(* Logix 5000 project; controller Drives_Line1 1756-L72 rev 20.13; software revision 20.04; part 9 of 21 *)
(* tags used below, declared in another part *)
   IO_State_Pinch_2 : INT;
   IO_State_Tmp_Pinch_2 : INT;
   Pinchroll_2_EncRes : DINT;
   Pinchroll_2_FB_Count_Old : DINT;
   Pinchroll_2_Max_FB_Counts : DINT;
   Pinchroll_2_Rev_mm : REAL;
   Pinchroll_2_RPMPerMPS : REAL;
   TonRefOn : TIMER;
   zPinchroll_2_Max_rev : REAL;
   Bridle_01 : UDT_Bridle_3M;
   EntryCtrl : UDT_Control_Zone;
   In_Config : UDT_Config;
   LineCmd : UDT_Commands_Line;
   Out_Feedbacks : UDT_Fdbks;
   Out_Status : UDT_Status;
   Pinchroll_2 : UDT_Pinchroll;
   Pinchroll_2_FB_Difference : DINT;
   Pinchroll_2_FB_Update_Valid : BOOL;
   Pinchroll_2_FBCounts_mm : REAL;
   TaskInterval_ms : DINT;
   TestConfig_Pinchroll_2 : UDT_Config_Pinch;
   Unwinder_1 : UDT_Unwinder;
   Unwinder_2 : UDT_Unwinder;
   zConfigFromMaster : BOOL;
   zPi : REAL;
   zPinchroll_2_EncRes : DINT;
(* P13_Pinchroll_2, continued *)

ROUTINE R03_Drive_Interface   (* ladder *)
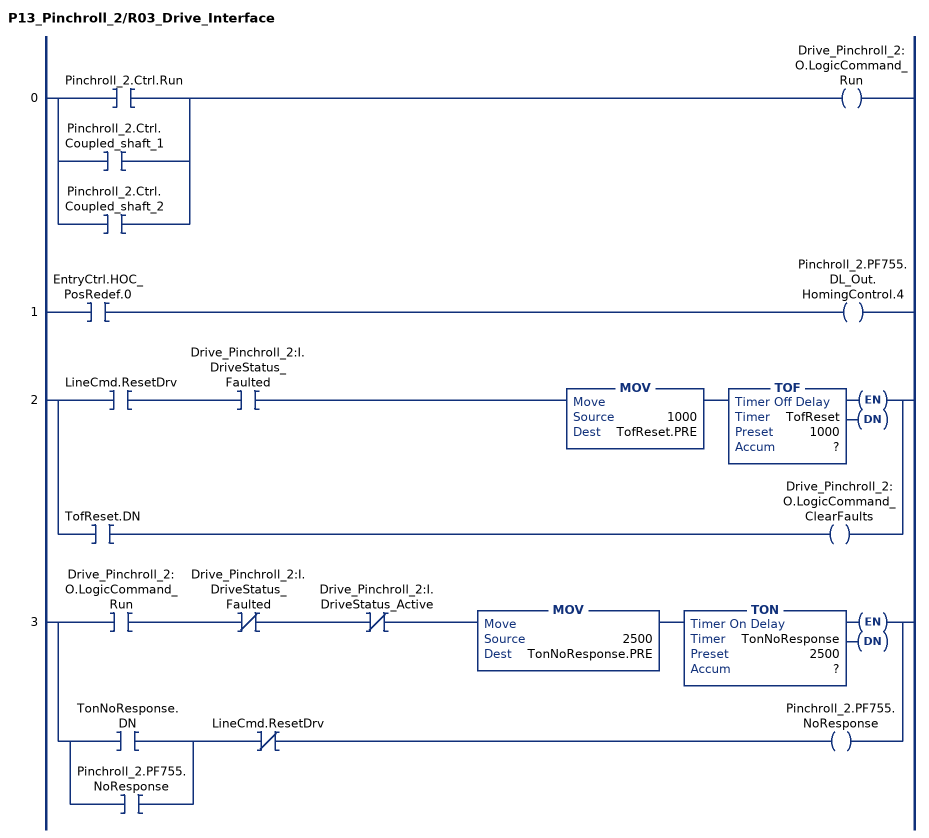
   0: [XIC(Pinchroll_2.Ctrl.Run) ,XIC(Pinchroll_2.Ctrl.Coupled_shaft_1) ,XIC(Pinchroll_2.Ctrl.Coupled_shaft_2) ]OTE(Drive_Pinchroll_2:O.LogicCommand_Run);
   1: XIC(EntryCtrl.HOC_PosRedef.0)OTE(Pinchroll_2.PF755.DL_Out.HomingControl.4);
   2: [XIC(LineCmd.ResetDrv) XIC(Drive_Pinchroll_2:I.DriveStatus_Faulted) MOV(1000,TofReset.PRE) TOF(TofReset,?,?) ,XIC(TofReset.DN) OTE(Drive_Pinchroll_2:O.LogicCommand_ClearFaults) ];
   3: [XIC(Drive_Pinchroll_2:O.LogicCommand_Run) XIO(Drive_Pinchroll_2:I.DriveStatus_Faulted) XIO(Drive_Pinchroll_2:I.DriveStatus_Active) MOV(2500,TonNoResponse.PRE) TON(TonNoResponse,?,?) ,[XIC(TonNoResponse.DN) ,XIC(Pinchroll_2.PF755.NoResponse) ] XIO(LineCmd.ResetDrv) OTE(Pinchroll_2.PF755.NoResponse) ];
END_ROUTINE

ROUTINE R04_State   (* ladder *)
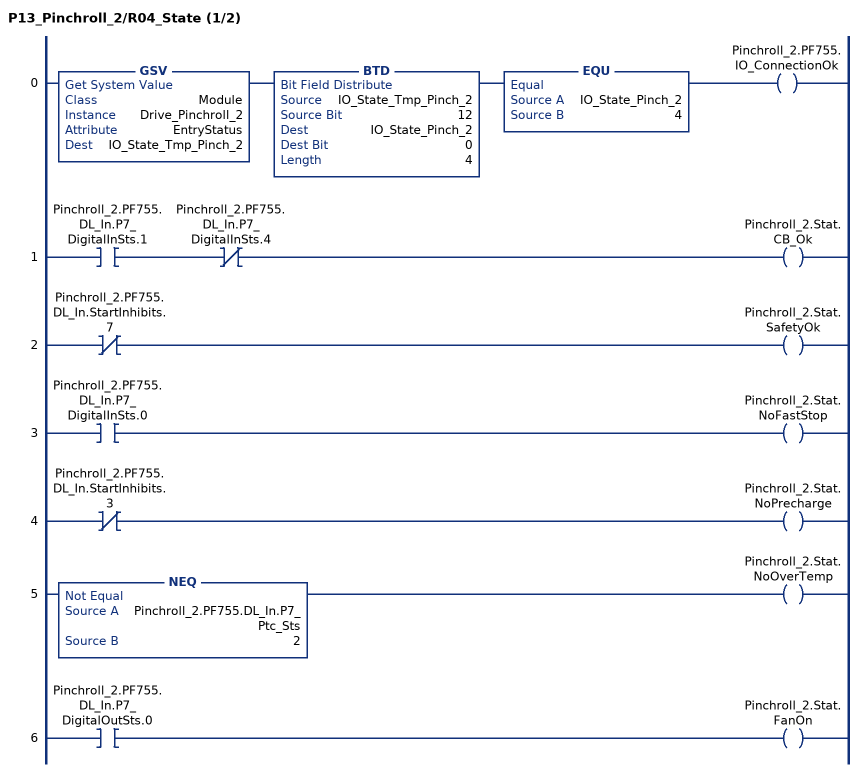
   0: GSV(Module,Drive_Pinchroll_2,EntryStatus,IO_State_Tmp_Pinch_2)BTD(IO_State_Tmp_Pinch_2,12,IO_State_Pinch_2,0,4)EQU(IO_State_Pinch_2,4)OTE(Pinchroll_2.PF755.IO_ConnectionOk);
   1: XIC(Pinchroll_2.PF755.DL_In.P7_DigitalInSts.1)XIO(Pinchroll_2.PF755.DL_In.P7_DigitalInSts.4)OTE(Pinchroll_2.Stat.CB_Ok);
   2: XIO(Pinchroll_2.PF755.DL_In.StartInhibits.7)OTE(Pinchroll_2.Stat.SafetyOk);
   3: XIC(Pinchroll_2.PF755.DL_In.P7_DigitalInSts.0)OTE(Pinchroll_2.Stat.NoFastStop);
   4: XIO(Pinchroll_2.PF755.DL_In.StartInhibits.3)OTE(Pinchroll_2.Stat.NoPrecharge);
   5: NEQ(Pinchroll_2.PF755.DL_In.P7_Ptc_Sts,2)OTE(Pinchroll_2.Stat.NoOverTemp);
   6: XIC(Pinchroll_2.PF755.DL_In.P7_DigitalOutSts.0)OTE(Pinchroll_2.Stat.FanOn);
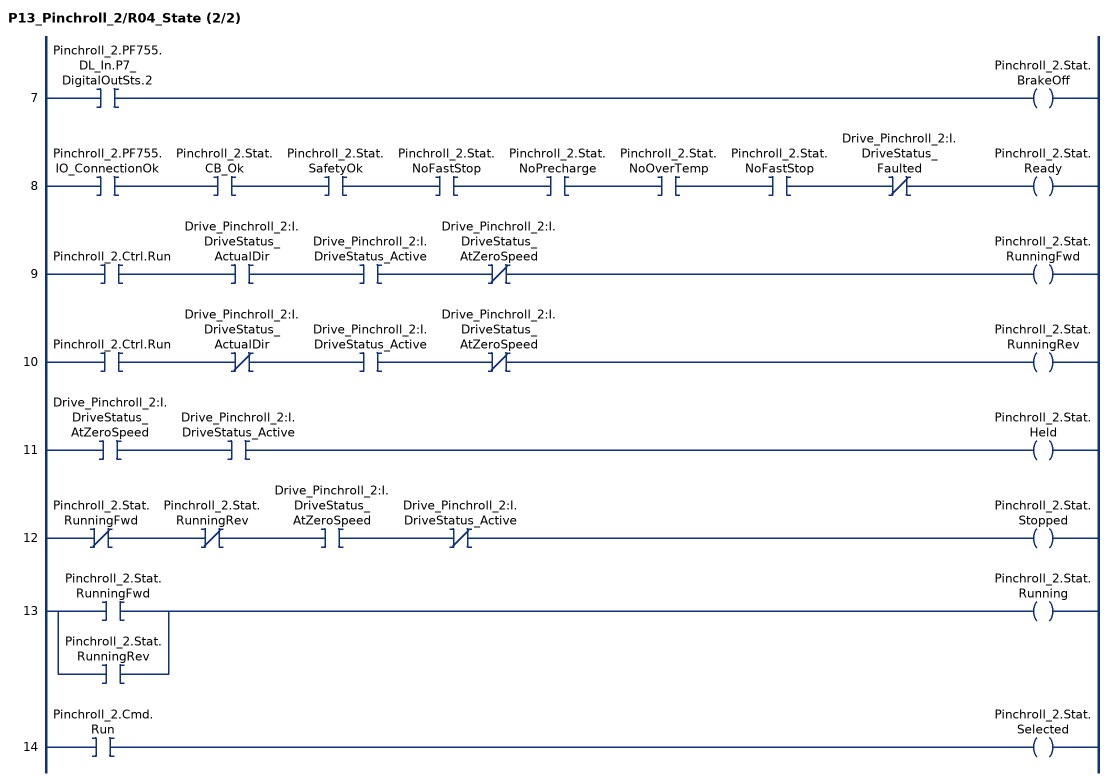
   7: XIC(Pinchroll_2.PF755.DL_In.P7_DigitalOutSts.2)OTE(Pinchroll_2.Stat.BrakeOff);
   8: XIC(Pinchroll_2.PF755.IO_ConnectionOk)XIC(Pinchroll_2.Stat.CB_Ok)XIC(Pinchroll_2.Stat.SafetyOk)XIC(Pinchroll_2.Stat.NoFastStop)XIC(Pinchroll_2.Stat.NoPrecharge)XIC(Pinchroll_2.Stat.NoOverTemp)XIC(Pinchroll_2.Stat.NoFastStop)XIO(Drive_Pinchroll_2:I.DriveStatus_Faulted)OTE(Pinchroll_2.Stat.Ready);
   9: XIC(Pinchroll_2.Ctrl.Run)XIC(Drive_Pinchroll_2:I.DriveStatus_ActualDir)XIC(Drive_Pinchroll_2:I.DriveStatus_Active)XIO(Drive_Pinchroll_2:I.DriveStatus_AtZeroSpeed)OTE(Pinchroll_2.Stat.RunningFwd);
   10: XIC(Pinchroll_2.Ctrl.Run)XIO(Drive_Pinchroll_2:I.DriveStatus_ActualDir)XIC(Drive_Pinchroll_2:I.DriveStatus_Active)XIO(Drive_Pinchroll_2:I.DriveStatus_AtZeroSpeed)OTE(Pinchroll_2.Stat.RunningRev);
   11: XIC(Drive_Pinchroll_2:I.DriveStatus_AtZeroSpeed)XIC(Drive_Pinchroll_2:I.DriveStatus_Active)OTE(Pinchroll_2.Stat.Held);
   12: XIO(Pinchroll_2.Stat.RunningFwd)XIO(Pinchroll_2.Stat.RunningRev)XIC(Drive_Pinchroll_2:I.DriveStatus_AtZeroSpeed)XIO(Drive_Pinchroll_2:I.DriveStatus_Active)OTE(Pinchroll_2.Stat.Stopped);
   13: [XIC(Pinchroll_2.Stat.RunningFwd) ,XIC(Pinchroll_2.Stat.RunningRev) ]OTE(Pinchroll_2.Stat.Running);
   14: XIC(Pinchroll_2.Cmd.Run)OTE(Pinchroll_2.Stat.Selected);
END_ROUTINE

ROUTINE R05_Control   (* ladder *)
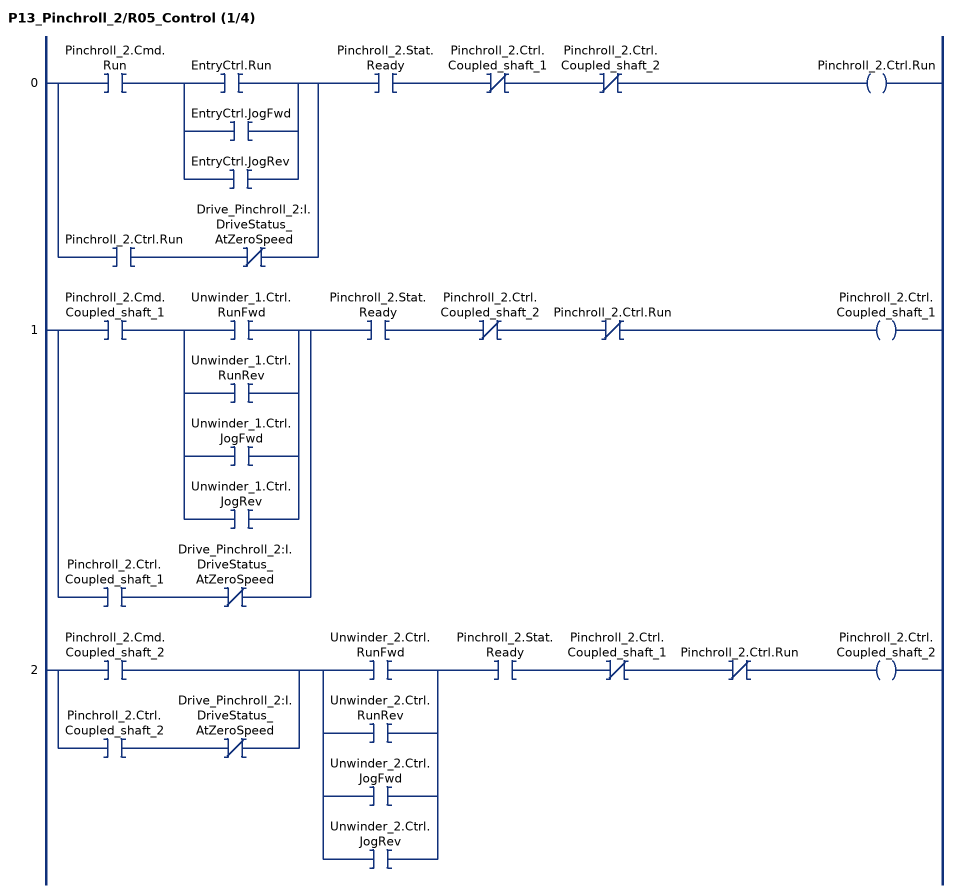
   0: [XIC(Pinchroll_2.Cmd.Run) [XIC(EntryCtrl.Run) ,XIC(EntryCtrl.JogFwd) ,XIC(EntryCtrl.JogRev) ] ,XIC(Pinchroll_2.Ctrl.Run) XIO(Drive_Pinchroll_2:I.DriveStatus_AtZeroSpeed) ]XIC(Pinchroll_2.Stat.Ready)XIO(Pinchroll_2.Ctrl.Coupled_shaft_1)XIO(Pinchroll_2.Ctrl.Coupled_shaft_2)OTE(Pinchroll_2.Ctrl.Run);
   1: [XIC(Pinchroll_2.Cmd.Coupled_shaft_1) [XIC(Unwinder_1.Ctrl.RunFwd) ,XIC(Unwinder_1.Ctrl.RunRev) ,XIC(Unwinder_1.Ctrl.JogFwd) ,XIC(Unwinder_1.Ctrl.JogRev) ] ,XIC(Pinchroll_2.Ctrl.Coupled_shaft_1) XIO(Drive_Pinchroll_2:I.DriveStatus_AtZeroSpeed) ]XIC(Pinchroll_2.Stat.Ready)XIO(Pinchroll_2.Ctrl.Coupled_shaft_2)XIO(Pinchroll_2.Ctrl.Run)OTE(Pinchroll_2.Ctrl.Coupled_shaft_1);
   2: [XIC(Pinchroll_2.Cmd.Coupled_shaft_2) ,XIC(Pinchroll_2.Ctrl.Coupled_shaft_2) XIO(Drive_Pinchroll_2:I.DriveStatus_AtZeroSpeed) ][XIC(Unwinder_2.Ctrl.RunFwd) ,XIC(Unwinder_2.Ctrl.RunRev) ,XIC(Unwinder_2.Ctrl.JogFwd) ,XIC(Unwinder_2.Ctrl.JogRev) ]XIC(Pinchroll_2.Stat.Ready)XIO(Pinchroll_2.Ctrl.Coupled_shaft_1)XIO(Pinchroll_2.Ctrl.Run)OTE(Pinchroll_2.Ctrl.Coupled_shaft_2);
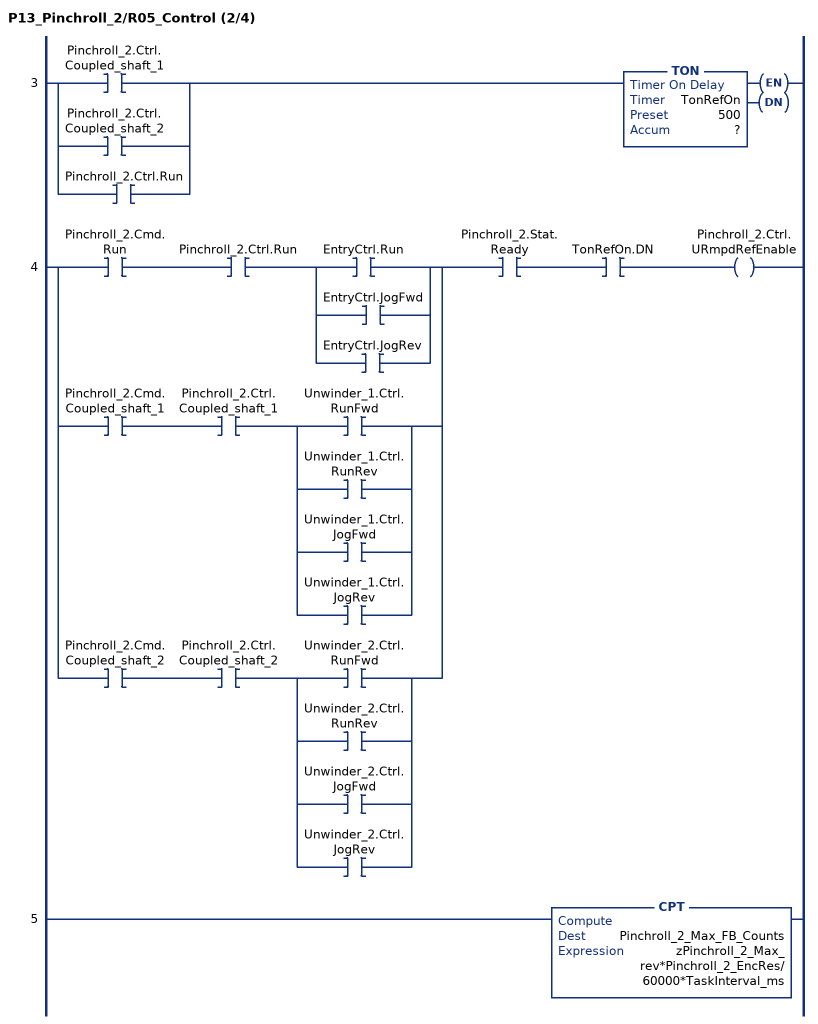
   3: [XIC(Pinchroll_2.Ctrl.Coupled_shaft_1) ,XIC(Pinchroll_2.Ctrl.Coupled_shaft_2) ,XIC(Pinchroll_2.Ctrl.Run) ]TON(TonRefOn,?,?);
   4: [XIC(Pinchroll_2.Cmd.Run) XIC(Pinchroll_2.Ctrl.Run) [XIC(EntryCtrl.Run) ,XIC(EntryCtrl.JogFwd) ,XIC(EntryCtrl.JogRev) ] ,XIC(Pinchroll_2.Cmd.Coupled_shaft_1) XIC(Pinchroll_2.Ctrl.Coupled_shaft_1) [XIC(Unwinder_1.Ctrl.RunFwd) ,XIC(Unwinder_1.Ctrl.RunRev) ,XIC(Unwinder_1.Ctrl.JogFwd) ,XIC(Unwinder_1.Ctrl.JogRev) ] ,XIC(Pinchroll_2.Cmd.Coupled_shaft_2) XIC(Pinchroll_2.Ctrl.Coupled_shaft_2) [XIC(Unwinder_2.Ctrl.RunFwd) ,XIC(Unwinder_2.Ctrl.RunRev) ,XIC(Unwinder_2.Ctrl.JogFwd) ,XIC(Unwinder_2.Ctrl.JogRev) ] ]XIC(Pinchroll_2.Stat.Ready)XIC(TonRefOn.DN)OTE(Pinchroll_2.Ctrl.URmpdRefEnable);
   5: CPT(Pinchroll_2_Max_FB_Counts,zPinchroll_2_Max_rev*Pinchroll_2_EncRes/60000*TaskInterval_ms);
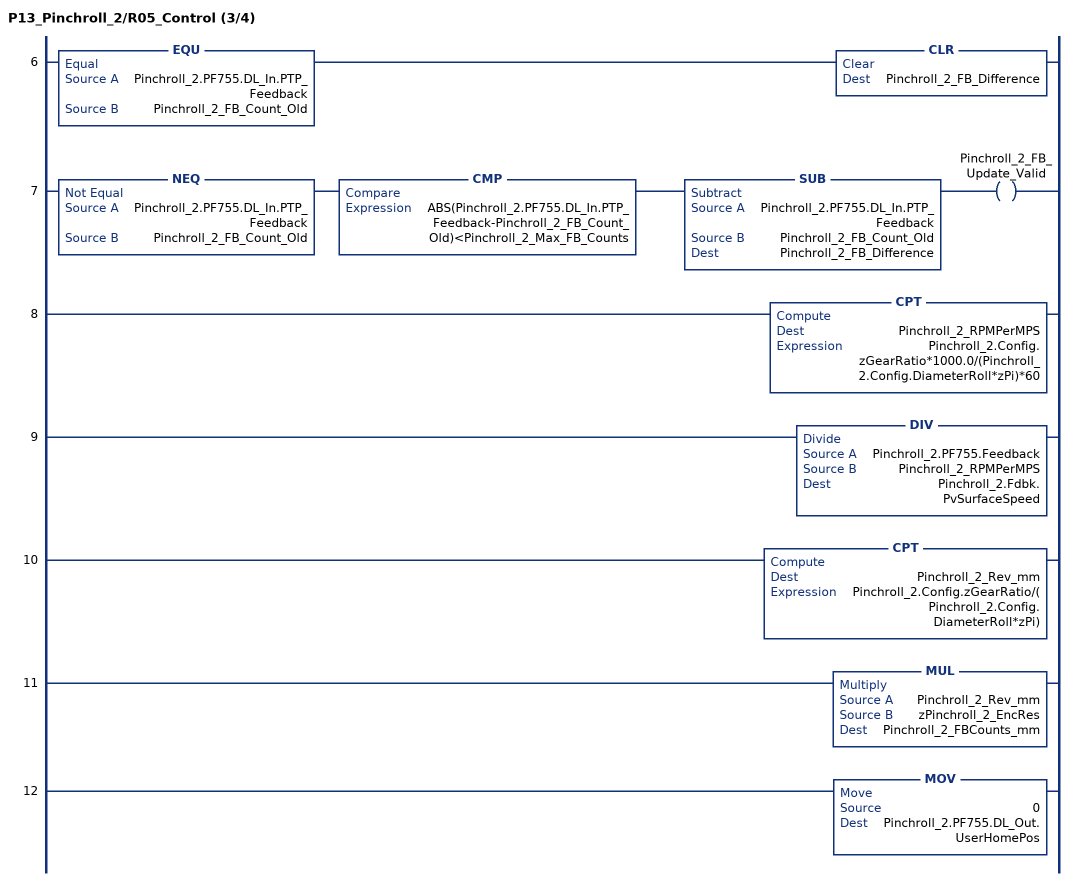
   6: EQU(Pinchroll_2.PF755.DL_In.PTP_Feedback,Pinchroll_2_FB_Count_Old)CLR(Pinchroll_2_FB_Difference);
   7: NEQ(Pinchroll_2.PF755.DL_In.PTP_Feedback,Pinchroll_2_FB_Count_Old)CMP(ABS(Pinchroll_2.PF755.DL_In.PTP_Feedback-Pinchroll_2_FB_Count_Old)<Pinchroll_2_Max_FB_Counts)SUB(Pinchroll_2.PF755.DL_In.PTP_Feedback,Pinchroll_2_FB_Count_Old,Pinchroll_2_FB_Difference)OTE(Pinchroll_2_FB_Update_Valid);
   8: CPT(Pinchroll_2_RPMPerMPS,Pinchroll_2.Config.zGearRatio*1000.0/(Pinchroll_2.Config.DiameterRoll*zPi)*60);
   9: DIV(Pinchroll_2.PF755.Feedback,Pinchroll_2_RPMPerMPS,Pinchroll_2.Fdbk.PvSurfaceSpeed);
   10: CPT(Pinchroll_2_Rev_mm,Pinchroll_2.Config.zGearRatio/(Pinchroll_2.Config.DiameterRoll*zPi));
   11: MUL(Pinchroll_2_Rev_mm,zPinchroll_2_EncRes,Pinchroll_2_FBCounts_mm);
   12: MOV(0,Pinchroll_2.PF755.DL_Out.UserHomePos);
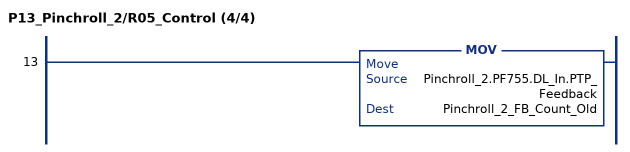
   13: MOV(Pinchroll_2.PF755.DL_In.PTP_Feedback,Pinchroll_2_FB_Count_Old);
END_ROUTINE

ROUTINE R12_DriveRef   (* function block diagram *)
   SHEET 1   // Select speed reference
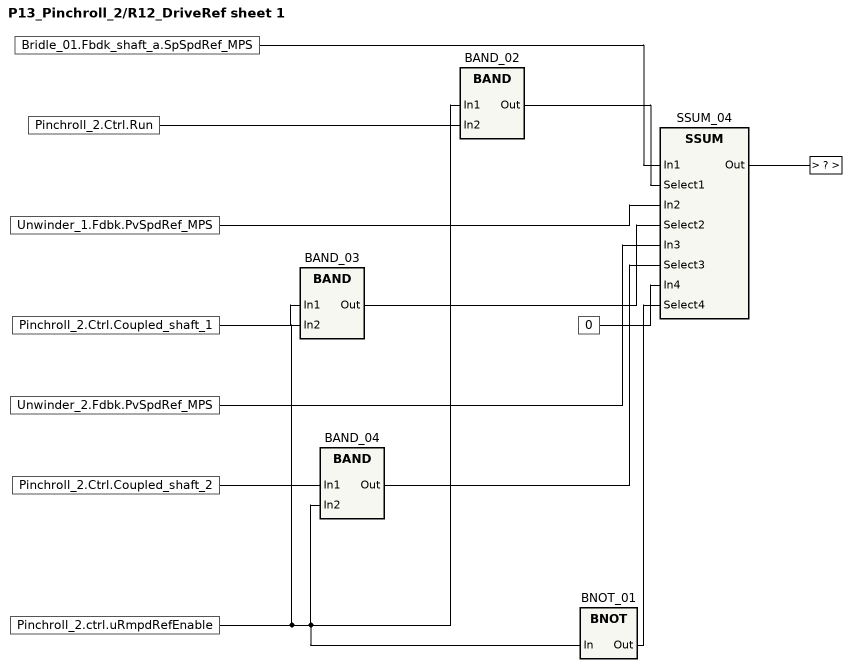
   BAND_03 : BAND(In1 := Pinchroll_2.Ctrl.Coupled_shaft_1, In2 := Pinchroll_2.ctrl.uRmpdRefEnable);
   BAND_04 : BAND(In1 := Pinchroll_2.Ctrl.Coupled_shaft_2, In2 := Pinchroll_2.ctrl.uRmpdRefEnable);
   BAND_02 : BAND(In1 := Pinchroll_2.ctrl.uRmpdRefEnable, In2 := Pinchroll_2.Ctrl.Run);
   BNOT_01 : BNOT(In := Pinchroll_2.ctrl.uRmpdRefEnable);
   SSUM_04 : SSUM(In1 := Bridle_01.Fbdk_shaft_a.SpSpdRef_MPS, Select1 := BAND_02.Out, In2 := Unwinder_1.Fdbk.PvSpdRef_MPS, Select2 := BAND_03.Out, In3 := Unwinder_2.Fdbk.PvSpdRef_MPS, Select3 := BAND_04.Out, In4 := 0, Select4 := BNOT_01.Out);
   WIRE(?) := SSUM_04.Out;
   SHEET 2   // Final speed reference
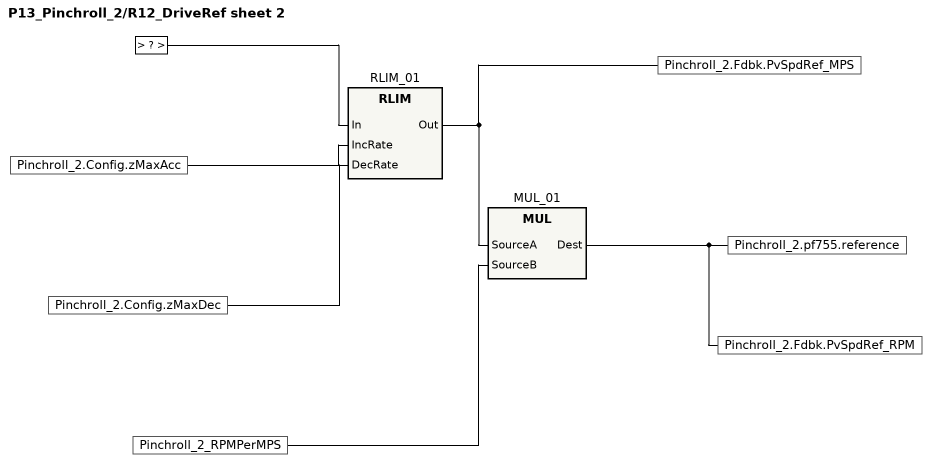
   RLIM_01 : RLIM(In := WIRE(?), IncRate := Pinchroll_2.Config.zMaxAcc, DecRate := Pinchroll_2.Config.zMaxDec);
   MUL_01 : MUL(SourceA := RLIM_01.Out, SourceB := Pinchroll_2_RPMPerMPS);
   Pinchroll_2.Fdbk.PvSpdRef_MPS := RLIM_01.Out;
   Pinchroll_2.Fdbk.PvSpdRef_RPM := MUL_01.Dest;
   Pinchroll_2.pf755.reference := MUL_01.Dest;
   SHEET 3   // Speed reference synchronized
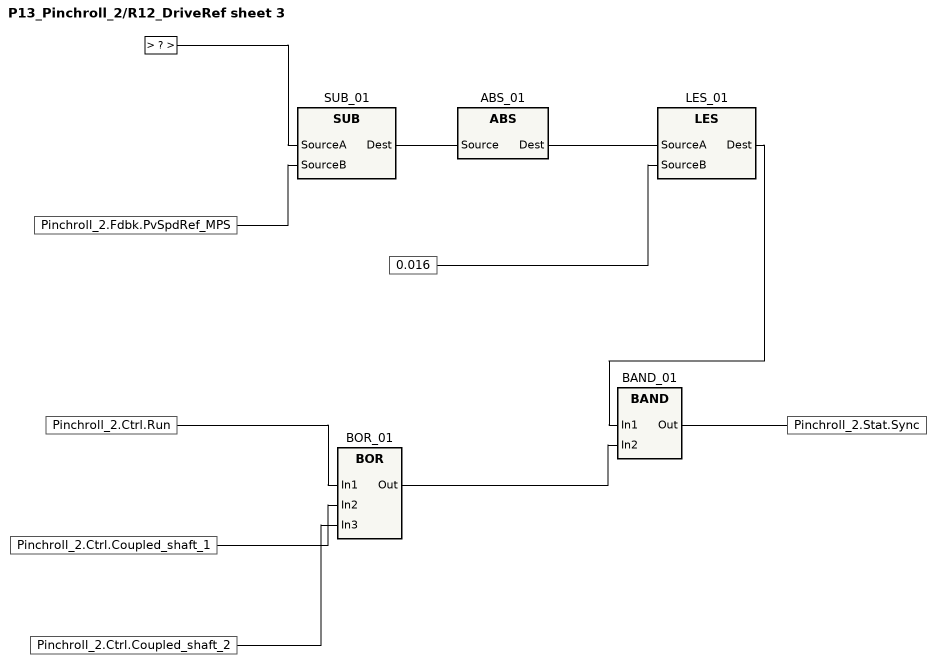
   SUB_01 : SUB(SourceA := WIRE(?), SourceB := Pinchroll_2.Fdbk.PvSpdRef_MPS);
   BOR_01 : BOR(In1 := Pinchroll_2.Ctrl.Run, In2 := Pinchroll_2.Ctrl.Coupled_shaft_1, In3 := Pinchroll_2.Ctrl.Coupled_shaft_2);
   ABS_01 : ABS(Source := SUB_01.Dest);
   LES_01 : LES(SourceA := ABS_01.Dest, SourceB := 0.016);
   BAND_01 : BAND(In1 := LES_01.Dest, In2 := BOR_01.Out);
   Pinchroll_2.Stat.Sync := BAND_01.Out;
END_ROUTINE

ROUTINE R98_ToDrive   (* ladder *)
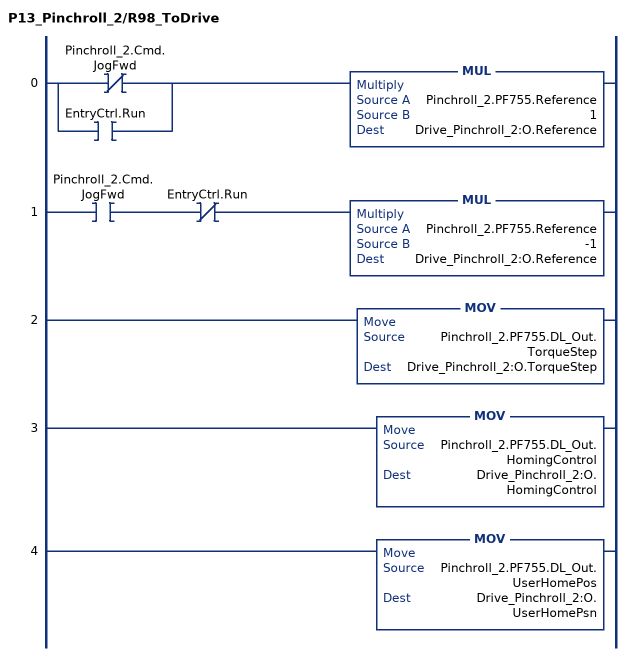
   0: [XIO(Pinchroll_2.Cmd.JogFwd) ,XIC(EntryCtrl.Run) ]MUL(Pinchroll_2.PF755.Reference,1,Drive_Pinchroll_2:O.Reference);
   1: XIC(Pinchroll_2.Cmd.JogFwd)XIO(EntryCtrl.Run)MUL(Pinchroll_2.PF755.Reference,-1,Drive_Pinchroll_2:O.Reference);
   2: MOV(Pinchroll_2.PF755.DL_Out.TorqueStep,Drive_Pinchroll_2:O.TorqueStep);
   3: MOV(Pinchroll_2.PF755.DL_Out.HomingControl,Drive_Pinchroll_2:O.HomingControl);
   4: MOV(Pinchroll_2.PF755.DL_Out.UserHomePos,Drive_Pinchroll_2:O.UserHomePsn);
END_ROUTINE

ROUTINE R999_Test   (* ladder *)
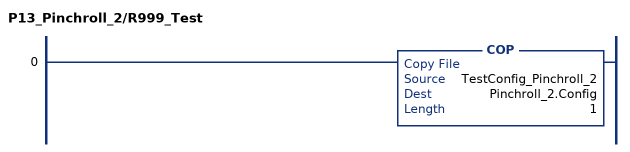
   0: COP(TestConfig_Pinchroll_2,Pinchroll_2.Config,1);
END_ROUTINE

ROUTINE R99_To_Master   (* ladder *)
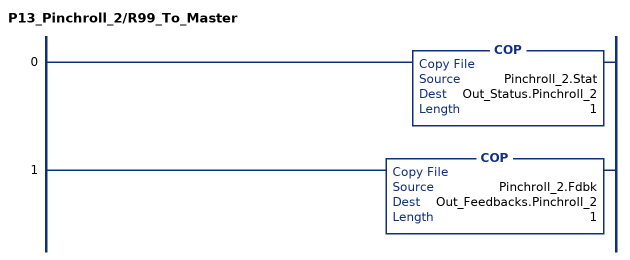
   0: COP(Pinchroll_2.Stat,Out_Status.Pinchroll_2,1);
   1: COP(Pinchroll_2.Fdbk,Out_Feedbacks.Pinchroll_2,1);
END_ROUTINE
END_PROGRAM

PROGRAM P14_Bridle_01   (* main routine R00_Main *)
VAR
   ADD_01 : FBD_MATH;
   BNOT_01 : FBD_BOOLEAN_NOT := (Out := 1);
   BNOT_02 : FBD_BOOLEAN_NOT := (In := 1);
   BNOT_03 : FBD_BOOLEAN_NOT := (Out := 1);
   Bridle_01_FB_Count_Old : DINT := 9220666;
   Bridle_01_Max_FBcounts : REAL := 5120.0;
   Bridle_01_SpdTrimMPS : REAL;
   Bridle_01_SpdTrimPct : REAL;
   Bridle_01a_RPMPerMPS : REAL := 3085.579;
   Bridle_01b_RPMPerMPS : REAL := 3085.579;
   Bridle_01c_RPMPerMPS : REAL := 2634.4192;
   DIV_01 : FBD_MATH := (SourceB := 100.0);
   EQU_01 : FBD_COMPARE := (SourceA := 0.08467744);
   IO_State_Bridle_01a : INT := 4;
   IO_State_Bridle_01b : INT := 4;
   IO_State_Bridle_01c : INT := 4;
   IO_State_Tmp_Bridle_01a : INT := 16384;
   IO_State_Tmp_Bridle_01b : INT := 16384;
   IO_State_Tmp_Bridle_01c : INT := 16384;
   MUL_01 : FBD_MATH := (SourceB := 3085.579);
   MUL_02 : FBD_MATH := (SourceB := 3085.579);
   MUL_05 : FBD_MATH;
   MUL_06 : FBD_MATH := (SourceB := 2634.4192);
   Ons : DINT;
   PI_02 : PROP_INT := (In := -2.3841858e-07, Initialize := 1, Kp := 0.1, Wld := 0.01, HighLimit := 2.5, LowLimit := -2.5, ShapeKpPlus := 1.0, ShapeKpMinus := 1.0, ShapeWldPlus := 1.0, ShapeWldMinus := 1.0, RTSTime := 1, DeltaT := 0.05);
   PulsReset_PID : TIMER := (PRE := 250);
   SCL_09 : SCALE := (InRawMax := 100.0, InRawMin := -100.0, InEUMax := 2.5, InEUMin := -2.5, Limiting := 1, Out := -2.3841858e-07);
   SUB_02 : FBD_MATH;
   TimeOn_PIDOn : TIMER := (PRE := 500);
   TofReset : TIMER := (PRE := 1000, ACC := 1000);
   TonNoResponse : TIMER[3] := ([0].PRE := 2500, [1].PRE := 2500, [2].PRE := 2500);
   zBridle_01_Ki_SpdTrim : REAL := 0.01;
   zBridle_01_Kp_SpdTrim : REAL := 0.1;
   zBridle_01_Max_rev : DINT := 1500;
   zBridle_01_MaxTrimSpdTrim : REAL := 2.5;
   zBridle_01_MinTrimSpdTrim : REAL := -2.5;
   zBridle_01b_EncRes : REAL := 4096.0;
END_VAR

ROUTINE R00_Main   (* ladder *)
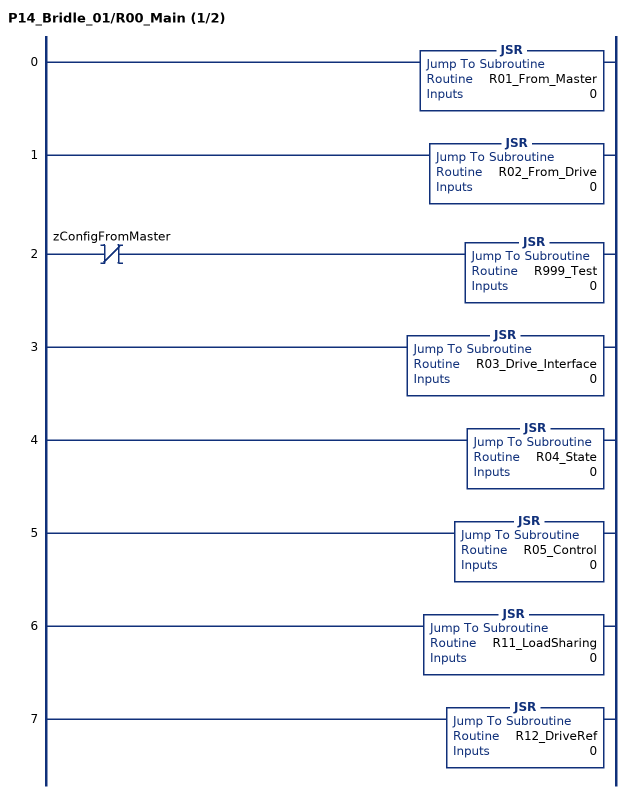
   0: JSR(R01_From_Master,0);
   1: JSR(R02_From_Drive,0);
   2: XIO(zConfigFromMaster)JSR(R999_Test,0);
   3: JSR(R03_Drive_Interface,0);
   4: JSR(R04_State,0);
   5: JSR(R05_Control,0);
   6: JSR(R11_LoadSharing,0);
   7: JSR(R12_DriveRef,0);
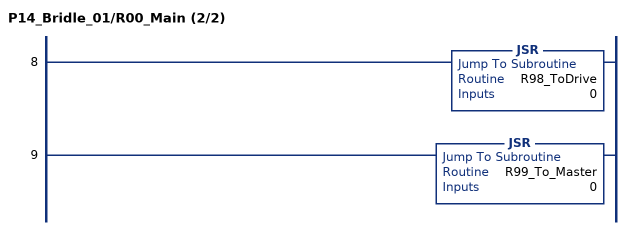
   8: JSR(R98_ToDrive,0);
   9: JSR(R99_To_Master,0);
END_ROUTINE

ROUTINE R01_From_Master   (* ladder *)
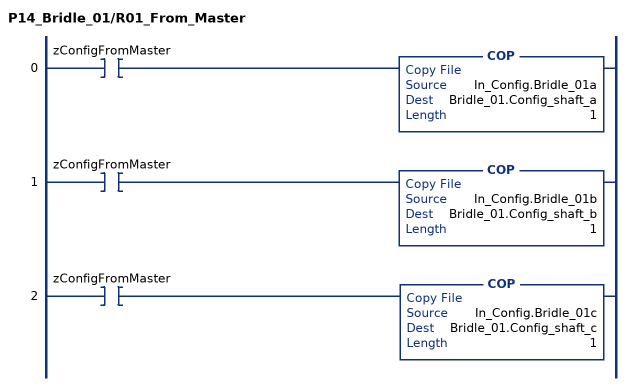
   0: XIC(zConfigFromMaster)COP(In_Config.Bridle_01a,Bridle_01.Config_shaft_a,1);
   1: XIC(zConfigFromMaster)COP(In_Config.Bridle_01b,Bridle_01.Config_shaft_b,1);
   2: XIC(zConfigFromMaster)COP(In_Config.Bridle_01c,Bridle_01.Config_shaft_c,1);
END_ROUTINE

ROUTINE R02_From_Drive   (* ladder *)
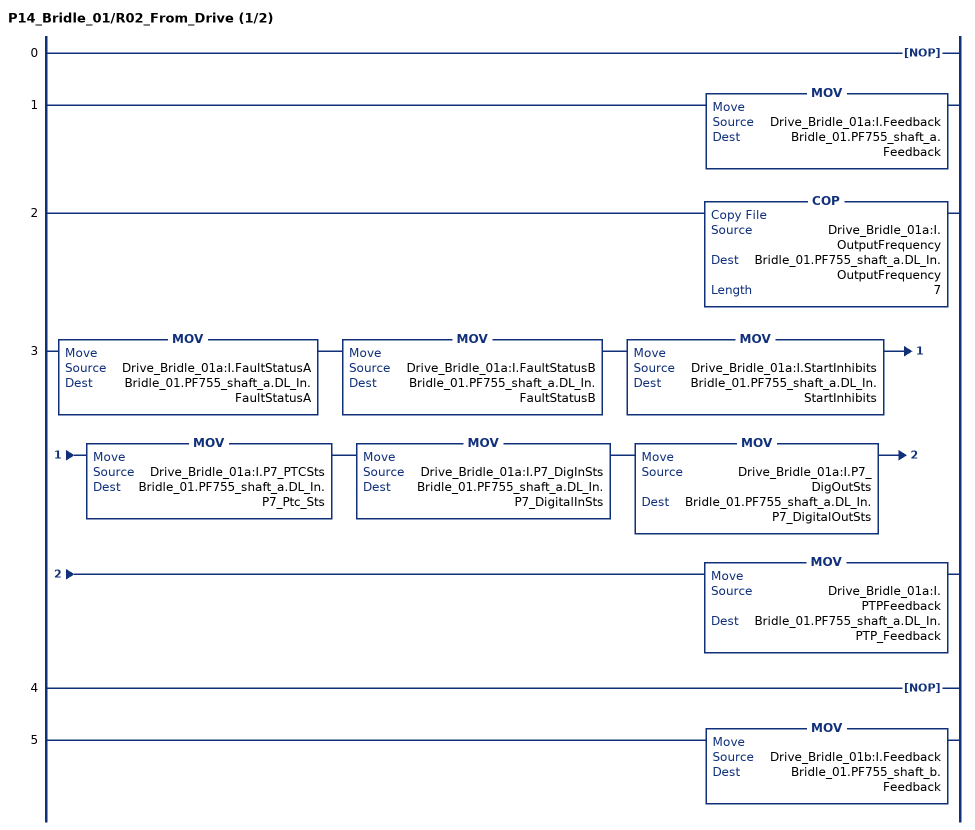
   0: NOP();
   1: MOV(Drive_Bridle_01a:I.Feedback,Bridle_01.PF755_shaft_a.Feedback);
   2: COP(Drive_Bridle_01a:I.OutputFrequency,Bridle_01.PF755_shaft_a.DL_In.OutputFrequency,7);
   3: MOV(Drive_Bridle_01a:I.FaultStatusA,Bridle_01.PF755_shaft_a.DL_In.FaultStatusA)MOV(Drive_Bridle_01a:I.FaultStatusB,Bridle_01.PF755_shaft_a.DL_In.FaultStatusB)MOV(Drive_Bridle_01a:I.StartInhibits,Bridle_01.PF755_shaft_a.DL_In.StartInhibits)MOV(Drive_Bridle_01a:I.P7_PTCSts,Bridle_01.PF755_shaft_a.DL_In.P7_Ptc_Sts)MOV(Drive_Bridle_01a:I.P7_DigInSts,Bridle_01.PF755_shaft_a.DL_In.P7_DigitalInSts)MOV(Drive_Bridle_01a:I.P7_DigOutSts,Bridle_01.PF755_shaft_a.DL_In.P7_DigitalOutSts)MOV(Drive_Bridle_01a:I.PTPFeedback,Bridle_01.PF755_shaft_a.DL_In.PTP_Feedback);
   4: NOP();
   5: MOV(Drive_Bridle_01b:I.Feedback,Bridle_01.PF755_shaft_b.Feedback);
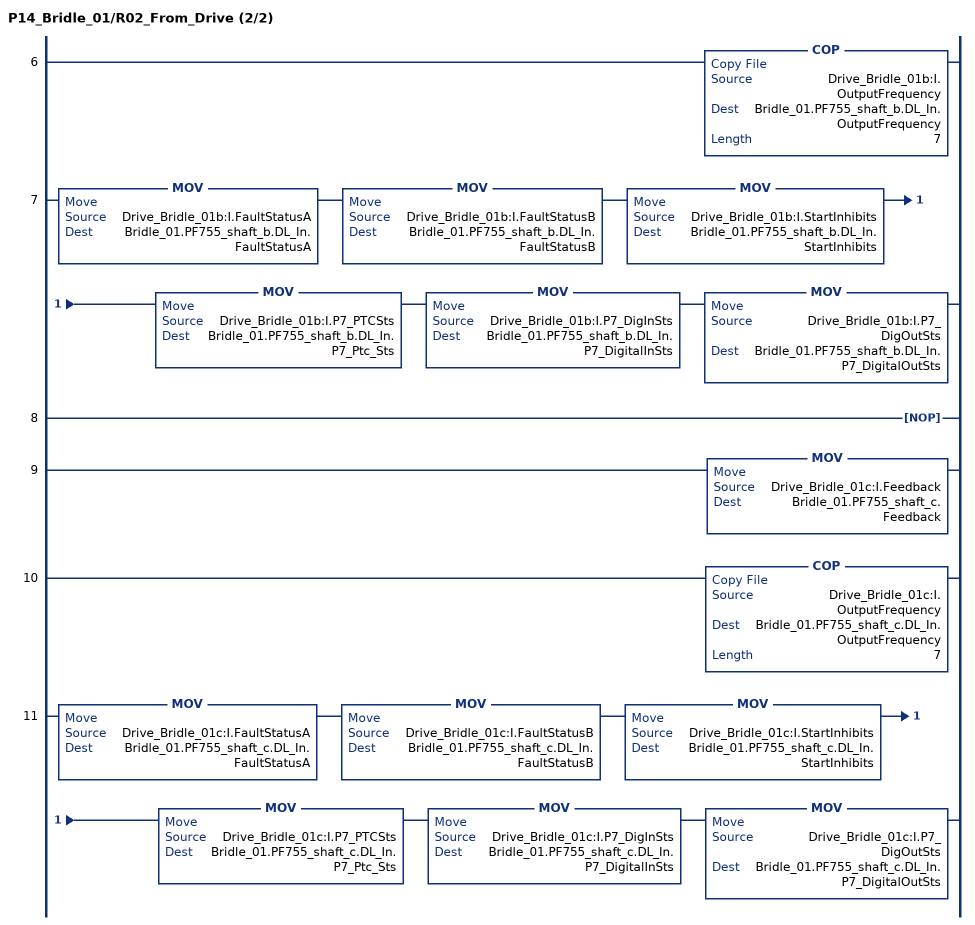
   6: COP(Drive_Bridle_01b:I.OutputFrequency,Bridle_01.PF755_shaft_b.DL_In.OutputFrequency,7);
   7: MOV(Drive_Bridle_01b:I.FaultStatusA,Bridle_01.PF755_shaft_b.DL_In.FaultStatusA)MOV(Drive_Bridle_01b:I.FaultStatusB,Bridle_01.PF755_shaft_b.DL_In.FaultStatusB)MOV(Drive_Bridle_01b:I.StartInhibits,Bridle_01.PF755_shaft_b.DL_In.StartInhibits)MOV(Drive_Bridle_01b:I.P7_PTCSts,Bridle_01.PF755_shaft_b.DL_In.P7_Ptc_Sts)MOV(Drive_Bridle_01b:I.P7_DigInSts,Bridle_01.PF755_shaft_b.DL_In.P7_DigitalInSts)MOV(Drive_Bridle_01b:I.P7_DigOutSts,Bridle_01.PF755_shaft_b.DL_In.P7_DigitalOutSts);
   8: NOP();
   9: MOV(Drive_Bridle_01c:I.Feedback,Bridle_01.PF755_shaft_c.Feedback);
   10: COP(Drive_Bridle_01c:I.OutputFrequency,Bridle_01.PF755_shaft_c.DL_In.OutputFrequency,7);
   11: MOV(Drive_Bridle_01c:I.FaultStatusA,Bridle_01.PF755_shaft_c.DL_In.FaultStatusA)MOV(Drive_Bridle_01c:I.FaultStatusB,Bridle_01.PF755_shaft_c.DL_In.FaultStatusB)MOV(Drive_Bridle_01c:I.StartInhibits,Bridle_01.PF755_shaft_c.DL_In.StartInhibits)MOV(Drive_Bridle_01c:I.P7_PTCSts,Bridle_01.PF755_shaft_c.DL_In.P7_Ptc_Sts)MOV(Drive_Bridle_01c:I.P7_DigInSts,Bridle_01.PF755_shaft_c.DL_In.P7_DigitalInSts)MOV(Drive_Bridle_01c:I.P7_DigOutSts,Bridle_01.PF755_shaft_c.DL_In.P7_DigitalOutSts);
END_ROUTINE
